TYPE SensorOutput :
STRUCT
	SensorName : STRING;
	SensorActive : BOOL;
	
	OutputType : STRING;
	OutputDescription : STRING;
	//OutputINT : INT;
	OutputBOOL : BOOL;
	//OutputREAL : REAL;
END_STRUCT
END_TYPE

(* stored: Version 1.1.0.1
   DUT SensorOutput: Id {fe4f6c8f-82f6-4c5f-9b4c-0111606a76b7} *)
